(* CODESYS project Kompresszor

Project tree, tasks and I/O mapping:
  Device : CODESYS Control Win V3, 3S - Smart Software Solutions GmbH, version 3.5.17.0
    Ethernet : Ethernet, 3S - Smart Software Solutions GmbH, version 3.5.17.0
      ModbusTCP_Slave_Device : ModbusTCP Slave Device, 3S - Smart Software Solutions GmbH, version 3.5.17.0
          settings: StartAdresses.HoldingRegister = 20; StartAdresses.InputRegister = 20
          unmapped channels: %IW20 Holding Registers, %QW20 Input Registers
  libraries: Standard, * (System)
  global variables GVL
  hibak/
    hibak_al/
    program prgHibak_Main [ST]
    program prgNemIndul [ST]
    program prgUzemido_tullep [ST]
  global variables I
  data type kompresszor
  program MANUAL_TEST [ST]
  program PLC_PRG [ST]
  program prgHiba_kijelzes [ST]
  program prgHiba_nem_megfelelo_komp_szam [ST]
  program prgHiba_Nyomas [ST]
  program prgHiba_stuck_at_0 [ST]
  program prgHiba_stuck_at_1 [ST]
  program prgLampak [ST]
  program prgLealitast [ST]
  program prgMozgoKompJavitas [ST]
  program prgNincs_eleg_komp [ST]
  program prgNyomas [ST]
  global variables Q
  program prgInditas [ST]
  program prgKompresszorok_szama [ST]
  program prgTiltas [ST]
  program prgUzemido [ST]
  task MainTask (cyclic, interval t#20ms, priority 1) calls input_led, MANUAL_TEST, PLC_PRG
*)

// kompresszor
TYPE kompresszor :
STRUCT
	tUzemido: TIME;
	xHiba: BOOL;
	xRun: BOOL;
END_STRUCT
END_TYPE

// GVL
{attribute 'qualified_only'}
VAR_GLOBAL
	start_r_trig: R_TRIG;
	start_f_trig: F_TRIG;
	stop_r_trig: R_TRIG;
	stop_f_trig: F_TRIG;
	emerg_r_trig: R_TRIG;
	emerg_f_trig: F_TRIG;
	
	komp1: oKompresszor;
	komp2: oKompresszor;
	komp3: oKompresszor;
	komp4: oKompresszor;
	
	tFelbontas: TIME := T#100MS;
	
	iKomp_Szuks: INT;
END_VAR

// I
{attribute 'qualified_only'}
VAR_GLOBAL
	ON AT %IX40.0 : BOOL;
	K1 AT %IX40.1 : BOOL;
	K2 AT %IX40.2 : BOOL;
	K3 AT %IX40.3 : BOOL;
	K4 AT %IX40.4 : BOOL;
	K1T AT %IX40.5 : BOOL;
	K2T AT %IX40.6 : BOOL;
	K3T AT %IX40.7 : BOOL;
	K4T AT %IX42.0 : BOOL;
	K1NJ AT %IX42.1 : BOOL;
	K2NJ AT %IX42.2 : BOOL;
	K3NJ AT %IX42.3 : BOOL;
	K4NJ AT %IX42.4 : BOOL;
	PMIN AT %IX42.5 : BOOL;
	PMID AT %IX42.6 : BOOL;
	PMAX AT %IX42.7 : BOOL;
END_VAR

// Q
{attribute 'qualified_only'}
VAR_GLOBAL
	K1 AT %QX40.0 : BOOL;
	K2 AT %QX40.1 : BOOL;
	K3 AT %QX40.2 : BOOL;
	K4 AT %QX40.3 : BOOL;
	K1L AT %QX40.4 : BOOL;
	K2L AT %QX40.5 : BOOL;
	K3L AT %QX40.6 : BOOL;
	K4L AT %QX40.7 : BOOL;
	HORN AT %QX41.0 : BOOL;
	ERR1 AT %QX41.1 : BOOL;
	ERR2 AT %QX41.2 : BOOL;
	ERR3 AT %QX41.3: BOOL;
	ERR4 AT %QX41.4 : BOOL;
	ERR5 AT %QX41.5 : BOOL;
	ERR6 AT %QX41.6 : BOOL;
	OPERATE AT %QX41.7 : BOOL;
	

	
END_VAR

// MANUAL_TEST
PROGRAM MANUAL_TEST
VAR
END_VAR

//KONZOL MUKODTETI AZ OUTPUTOKAT
%QW20 := %IW5;

END_PROGRAM

// PLC_PRG
PROGRAM PLC_PRG
VAR
END_VAR

GVL.start_r_trig(CLK:= I.ON);
GVL.start_f_trig(CLK:= I.ON);
// GVL.stop_r_trig(CLK:= I.STOP_NC);
// GVL.stop_f_trig(CLK:= I.STOP_NC);
// GVL.emerg_r_trig(CLK:= I.EMERG_NC);
// GVL.emerg_f_trig(CLK:= I.EMERG_NC);
GVL.K1NJ_r_trig(CLK:= I.K1NJ);
GVL.K2NJ_r_trig(CLK:= I.K2NJ);
GVL.K3NJ_r_trig(CLK:= I.K3NJ);
GVL.K4NJ_r_trig(CLK:= I.K4NJ);

END_PROGRAM

// prgHiba_kijelzes
PROGRAM prgHiba_kijelzes
VAR
END_VAR

q.ERR1 := prgHiba_Nyomas.hiba;
// q.ERR2 := ;
q.ERR3 := prgNincs_eleg_komp.hiba;
q.ERR4 := prgMozgoKompJavitas.hiba;
q.ERR5 := prgHiba_nem_megfelelo_komp_szam.hiba;
// q.ERR4 :=

END_PROGRAM

// prgHiba_Nyomas
PROGRAM prgHiba_Nyomas
VAR
	hiba :BOOL;
END_VAR

IF 
	(NOT I.PMID AND I.PMAX) OR
	(NOT I.PMIN AND I.PMID)
THEN
	hiba := TRUE;
END_IF

END_PROGRAM

// prgNincs_eleg_komp
PROGRAM prgNincs_eleg_komp
VAR
	HIBAS_komp :INT;
	hiba :BOOL;
END_VAR

HIBAS_komp := BOOL_TO_INT(KOMP1.XHIBA) + BOOL_TO_INT(KOMP2.XHIBA) + BOOL_TO_INT(KOMP3.XHIBA) + BOOL_TO_INT(KOMP4.XHIBA);

//hiba ha nincs eleg komp
IF gvl.iKomp_Szuks <= (4 - HIBAS_komp) THEN
	hiba := FALSE;
ELSE
	hiba := TRUE;
END_IF

END_PROGRAM

// prgMozgoKompJavitas
PROGRAM prgMozgoKompJavitas
VAR
	hiba :BOOL;
END_VAR

IF
	i.K1 AND i.K1NJ OR
	i.K2 AND i.K2NJ OR
	i.K3 AND i.K3NJ OR
	i.K4 AND i.K4NJ
THEN
	hiba := TRUE;
ELSE
	hiba := FALSE;
END_IF

END_PROGRAM

// prgHiba_nem_megfelelo_komp_szam
PROGRAM prgHiba_nem_megfelelo_komp_szam
VAR
	hiba :BOOL;
	mukodo_komp :INT;
END_VAR

mukodo_komp := BOOL_TO_INT(I.K1) + BOOL_TO_INT(I.K2) + BOOL_TO_INT(I.K3) + BOOL_TO_INT(I.K4);

IF GVL.iKomp_Szuks <> mukodo_komp THEN
	HIBA:=TRUE;
ELSE
	HIBA := FALSE;	
END_IF

END_PROGRAM

// prgHiba_stuck_at_0
PROGRAM prgHiba_stuck_at_0
VAR
END_VAR

END_PROGRAM

// prgHiba_stuck_at_1
PROGRAM prgHiba_stuck_at_1
VAR
END_VAR

END_PROGRAM

// prgLampak
PROGRAM prgLampak
VAR
	villogo1 :fbBlinker2;
	villogo2 :fbBlinker2;
	villogo3 :fbBlinker2;
	villogo4 :fbBlinker2;
	time_on : TIME:= T#500MS;
	time_of : TIME:= T#500MS;	
END_VAR

// LAMPAK 
// 1 KOMPRESSZOR
IF gvl.komp1.xRun THEN
	q.K1L := TRUE;
ELSIF gvl.komp1.xHiba THEN
	q.K1L := villogo1.Q;
ELSE
	q.K1L := FALSE;
END_IF
//2 KOMPRESSZOR
IF gvl.komp2.xRun THEN
	q.K2L := TRUE;
ELSIF gvl.komp2.xHiba THEN
	q.K2L := villogo2.Q;
ELSE
	q.K2L := FALSE;
END_IF
// 3 KOMPRESSZOR
IF gvl.komp3.xRun THEN
	q.K3L := TRUE;
ELSIF gvl.komp3.xHiba THEN
	q.K3L := villogo3.Q;
ELSE
	q.K3L := FALSE;
END_IF
// 4 KOMPRESSZOR 
IF gvl.komp4.xRun THEN
	q.K4L := TRUE;
ELSIF gvl.komp4.xHiba THEN
	q.K4L := villogo4.Q;
ELSE
	q.K4L := FALSE;
END_IF

villogo1(ENABLE := gvl.komp1.xRun ,time_on := time_on , TIME_OFF :=time_of );
villogo2(ENABLE := gvl.komp2.xRun ,time_on := time_on , TIME_OFF :=time_of );
villogo3(ENABLE := gvl.komp3.xRun ,time_on := time_on , TIME_OFF :=time_of );
villogo4(ENABLE := gvl.komp4.xRun ,time_on := time_on , TIME_OFF :=time_of );

END_PROGRAM

// prgLealitast
PROGRAM prgLealitast
VAR
END_VAR

END_PROGRAM

// prgNyomas
PROGRAM prgNyomas
VAR
	komp_szam
END_VAR

END_PROGRAM

// hibak/prgHibak_Main
PROGRAM prgHibak_Main
VAR
END_VAR

prgHiba_kijelzes();

prgHiba_nem_megfelelo_komp_szam();
prgHiba_Nyomas();
prgMozgoKompJavitas();
prgNincs_eleg_komp();
prgUzemido_tullep();
prgNemIndul();

END_PROGRAM

// hibak/prgUzemido_tullep
PROGRAM prgUzemido_tullep
VAR
	hiba :BOOL;
END_VAR

// IF
// 	AND I.K1 OR
// 	AND I.K2 OR
// 	AND I.K3 OR
// 	AND I.K4
// THEN
// 	hiba:= TRUE;
// ELSE
// 	hiba := FALSE;
// END_IF

END_PROGRAM

// hibak/prgNemIndul
PROGRAM prgNemIndul
VAR
	hiba : BOOL;
END_VAR

IF
	gvl.Hiba1 OR
	gvl.Hiba2 OR
	gvl.Hiba3 OR
	gvl.Hiba4
THEN
	HIBA:= TRUE;
ELSE
	HIBA:= FALSE;
END_IF

END_PROGRAM

// prgInditas
PROGRAM prgInditas
VAR
	aiKompUzemidok: ARRAY [0..3] OF INT;
	iLegkisebbUzemideju: INT;
	iJelenlegVizsgalt: INT;
END_VAR

aiKompUzemidok[0] := gvl.aoKompTomb[0].iUzemido;
aiKompUzemidok[1] := gvl.aoKompTomb[1].iUzemido;
aiKompUzemidok[2] := gvl.aoKompTomb[2].iUzemido;
aiKompUzemidok[3] := gvl.aoKompTomb[3].iUzemido;
iLegkisebbUzemideju := 0;
IF gvl.aoKompTomb[0].xHiba OR gvl.aoKompTomb[0].xRun THEN
	ilegkisebbuzemideju := 1;
END_IF

IF gvl.aoKompTomb[1].xHiba OR gvl.aoKompTomb[1].xRun THEN
	ilegkisebbuzemideju := 2;
END_IF

IF gvl.aoKompTomb[2].xHiba OR gvl.aoKompTomb[2].xRun THEN
	ilegkisebbuzemideju := 3;
END_IF

IF gvl.aoKompTomb[3].xHiba OR gvl.aoKompTomb[3].xRun THEN
	ilegkisebbuzemideju := 4;
END_IF

IF gvl.iKomp_Szuks > GVL.iKomp_Futok THEN
	FOR iJelenlegVizsgalt := (iLegkisebbUzemideju + 1) TO 4 DO
		IF aiKompUzemidok[iJelenlegVizsgalt] < aiKompUzemidok[iLegkisebbUzemideju] AND NOT aiKompUzemidok[iJelenlegVizsgalt].xrun  THEN
			iLegkisebbUzemideju := iJelenlegVizsgalt;
		END_IF
	END_FOR
	
	CASE iLegkisebbUzemideju OF
		0: gvl.aoKompTomb[0].xRun := TRUE;
		1: gvl.aoKompTomb[0].xRun := TRUE;
		2: gvl.aoKompTomb[1].xRun := TRUE;
		3: gvl.aoKompTomb[2].xRun := TRUE;
	END_CASE
END_IF

END_PROGRAM

// prgKompresszorok_szama
PROGRAM prgKompresszorok_szama
VAR
	iKompresszorok : int;
END_VAR

GVL.iKomp_Futok := 0;
GVL.iKomp_Hibasak := 0;

FOR iKompresszorok := 0 TO 4 DO
	IF GVL.aoKompTomb[iKompresszorok].xRun THEN
		GVL.iKomp_Futok := GVL.iKomp_Futok + 1;
	END_IF 
	IF GVL.aoKompTomb[iKompresszorok].xHiba THEN
		GVL.iKomp_Hibasak := GVL.iKomp_Hibasak + 1;
	END_IF 
END_FOR

END_PROGRAM

// prgTiltas
PROGRAM prgTiltas
VAR
	tK1 :ton;
	tK2 :ton;
	tK3 :ton;
	tK4 :ton;
END_VAR

IF i.K1T AND gvl.aoKompTomb[0].xRun THEN
	gvl.aoKompTomb[0].xRun :=FALSE;
END_IF

IF i.K2T AND gvl.aoKompTomb[1].xRun THEN
	gvl.aoKompTomb[1].xRun :=FALSE;
END_IF

IF i.K3T AND gvl.aoKompTomb[2].xRun THEN
	gvl.aoKompTomb[2].xRun :=FALSE;
END_IF

IF i.K4T AND gvl.aoKompTomb[3].xRun THEN
	gvl.aoKompTomb[3].xRun :=FALSE;
END_IF

gvl.aoKompTomb[0].xHiba := I.K1T OR (gvl.aoKompTomb[0].iUzemido = 3000);
gvl.aoKompTomb[1].xHiba := I.K2T OR (gvl.aoKompTomb[1].iUzemido = 3000);
gvl.aoKompTomb[2].xHiba := I.K3T OR (gvl.aoKompTomb[2].iUzemido = 3000);
gvl.aoKompTomb[3].xHiba := I.K4T OR (gvl.aoKompTomb[3].iUzemido = 3000);

IF tk1.Q AND NOT i.K1 THEN
	gvl.Hiba1 := TRUE;
END_IF
IF tk2.Q AND NOT i.K2 THEN
	gvl.Hiba2 := TRUE;
END_IF
IF tk3.Q AND NOT i.K3 THEN
	gvl.Hiba3 := TRUE;
END_IF
IF tk4.Q AND NOT i.K4 THEN
	gvl.Hiba4 := TRUE;
END_IF

tK1(IN:= gvl.aoKompTomb[0].xRun, PT:= T#500MS);
tK2(IN:= gvl.aoKompTomb[1].xRun, PT:= T#500MS);
tK3(IN:= gvl.aoKompTomb[2].xRun, PT:= T#500MS);
tK4(IN:= gvl.aoKompTomb[3].xRun, PT:= T#500MS);

END_PROGRAM

// prgUzemido
PROGRAM prgUzemido
VAR
	tonFelbontas: TON;
END_VAR

tonFelbontas(PT:= GVL.tFelbontas);

IF NOT tonFelbontas.IN THEN
	tonFelbontas.IN := TRUE;
END_IF

IF GVL.komp1.xRun AND tonFelbontas.Q THEN
	GVL.komp1.iUzemido := GVL.komp1.iUzemido + 1;
END_IF

IF GVL.komp2.xRun AND tonFelbontas.Q THEN
	GVL.komp2.iUzemido := GVL.komp2.iUzemido + 1;
END_IF

IF GVL.komp3.xRun AND tonFelbontas.Q THEN
	GVL.komp3.iUzemido := GVL.komp3.iUzemido + 1;
END_IF

IF GVL.komp4.xRun AND tonFelbontas.Q THEN
	GVL.komp4.iUzemido := GVL.komp4.iUzemido + 1;
END_IF

IF tonFelbontas.Q THEN
	tonFelbontas.IN := FALSE;
END_IF

END_PROGRAM
